Fanuc KAREL source: kt00186.KL

PROGRAM KT00186
%NOLOCKGROUP
VAR
H1 : ARRAY[2] OF SHORT
I2:INTEGER
OUT:REAL
BEGIN
H1[1]=2
I2=3
OUT=((H1[1] MOD I2))
END KT00186
